(* PLC project extended wxHMI example, Unknown Beremiz 1 *)
(* stored: creationDateTime 2012-09-12T23:30:19, modificationDateTime 2018-09-26T14:07:02 *)

FUNCTION_BLOCK clock
  VAR
    TimerOn : TON;
  END_VAR
  VAR_OUTPUT
    Out : BOOL;
  END_VAR
  VAR_INPUT
    Period : TIME := T#3s;
  END_VAR
  VAR
    TimerOff : TON;
  END_VAR
  VAR  (* added by the conversion: wires and edge detectors of the diagram *)
    _DIV16_OUT : TIME;
  END_VAR

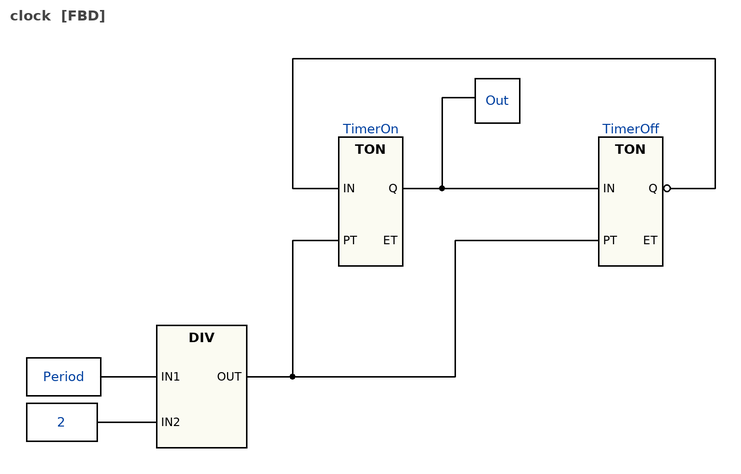
(* FBD diagram, written out as Structured Text *)
_DIV16_OUT := Period / 2;
TimerOff(IN := TimerOn.Q, PT := _DIV16_OUT);
TimerOn(IN := NOT TimerOff.Q, PT := _DIV16_OUT);
Out := TimerOn.Q;
END_FUNCTION_BLOCK

FUNCTION_BLOCK axis
  VAR_INPUT
    Power : BOOL;
    Up : BOOL;
    Down : BOOL;
  END_VAR
  VAR_OUTPUT
    Out : INT;
  END_VAR
  VAR
    axis_conuter : CTUD;
    clock0 : clock;
  END_VAR
  VAR  (* added by the conversion: wires and edge detectors of the diagram *)
    _AND4_OUT : BOOL;
    R_TRIG1 : R_TRIG;
    R_TRIG2 : R_TRIG;
  END_VAR

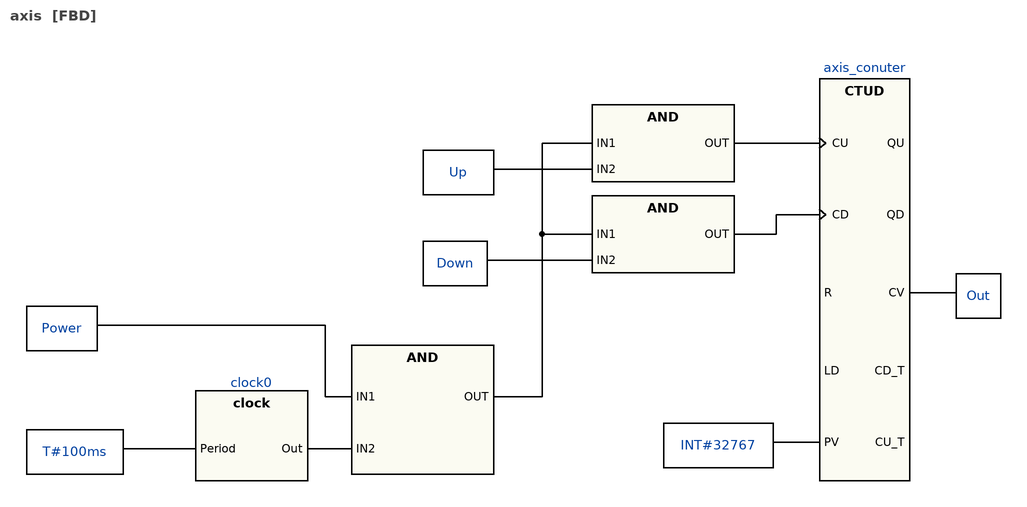
(* FBD diagram, written out as Structured Text *)
clock0(Period := T#100ms);
_AND4_OUT := Power AND clock0.Out;
R_TRIG1(CLK := _AND4_OUT AND Up);
R_TRIG2(CLK := _AND4_OUT AND Down);
axis_conuter(CU := R_TRIG1.Q, CD := R_TRIG2.Q, PV := INT#32767);
Out := axis_conuter.CV;
END_FUNCTION_BLOCK

PROGRAM main
  VAR_EXTERNAL
    Power_ON : BOOL;
    Power_OFF : BOOL;
  END_VAR
  VAR
    power : BOOL;
  END_VAR
  VAR_EXTERNAL
    DrawTest : BOOL;
    DrawTestBtn : BOOL;
    DrawLogo : BOOL;
    XaxisPos : INT;
    YaxisPos : INT;
    ZaxisPos : INT;
    TaxisPos : INT;
  END_VAR
  VAR
    PowerCtrl : RS;
    Xaxis : axis;
  END_VAR
  VAR_EXTERNAL
    XAxisMinus : BOOL;
    XAxisPlus : BOOL;
    YAxisPlus : BOOL;
    YAxisMinus : BOOL;
    ZAxisPlus : BOOL;
    ZAxisMinus : BOOL;
    TAxisPlus : BOOL;
    TAxisMinus : BOOL;
  END_VAR
  VAR
    Yaxis : axis;
    Taxis : axis;
    Zaxis : axis;
    DrawTestDo : RS;
    DrawLogoDo : RS;
  END_VAR

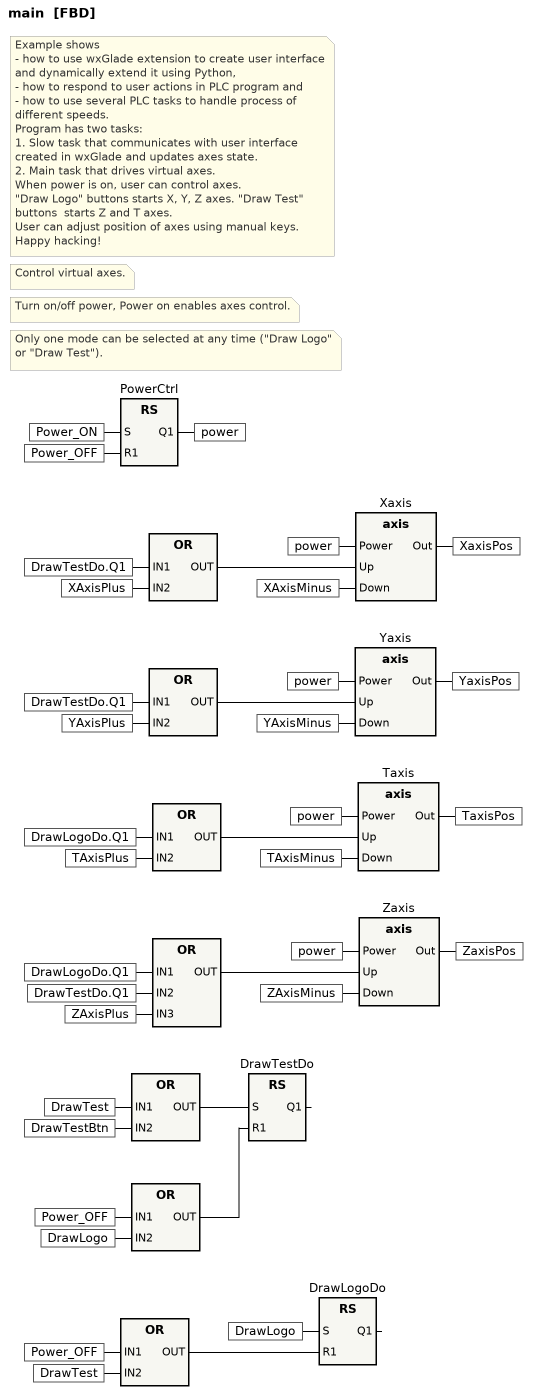
(* FBD diagram, written out as Structured Text *)
(* Example shows 
- how to use wxGlade extension to create user interface and dynamically extend it using Python, 
- how to respond to user actions in PLC program and 
- how to use several PLC tasks to handle process of different speeds.

Program has two tasks:
1. Slow task that communicates with user interface created in wxGlade and updates axes state.
2. Main task that drives virtual axes.

When power is on, user can control axes.
"Draw Logo" buttons starts X, Y, Z axes. "Draw Test" buttons  starts Z and T axes. 
User can adjust position of axes using manual keys.


Happy hacking! *)
(* Turn on/off power, Power on enables axes control. *)
PowerCtrl(S := Power_ON, R1 := Power_OFF);
power := PowerCtrl.Q1;
(* Only one mode can be selected at any time ("Draw Logo" or "Draw Test"). *)
(* Control virtual axes. *)
Xaxis(Power := power, Up := DrawTestDo.Q1 OR XAxisPlus, Down := XAxisMinus);
XaxisPos := Xaxis.Out;
Yaxis(Power := power, Up := DrawTestDo.Q1 OR YAxisPlus, Down := YAxisMinus);
YaxisPos := Yaxis.Out;
Zaxis(Power := power, Up := DrawLogoDo.Q1 OR DrawTestDo.Q1 OR ZAxisPlus, Down := ZAxisMinus);
ZaxisPos := Zaxis.Out;
Taxis(Power := power, Up := DrawLogoDo.Q1 OR TAxisPlus, Down := TAxisMinus);
TaxisPos := Taxis.Out;
DrawTestDo(S := DrawTest OR DrawTestBtn, R1 := Power_OFF OR DrawLogo);
DrawLogoDo(S := DrawLogo, R1 := Power_OFF OR DrawTest);
END_PROGRAM

PROGRAM ReadGUIdata
  VAR
    python_poll0 : python_poll;
  END_VAR

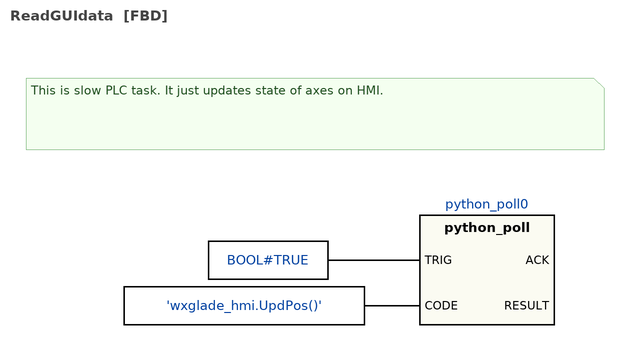
(* FBD diagram, written out as Structured Text *)
(* This is slow PLC task. It just updates state of axes on HMI. *)
python_poll0(TRIG := BOOL#TRUE, CODE := 'wxglade_hmi.UpdPos()');
END_PROGRAM

PROGRAM Declarations
  VAR
    InitValue : DINT := 17;
    NotInitializedVariable : DINT;
    counter : DINT;
  END_VAR

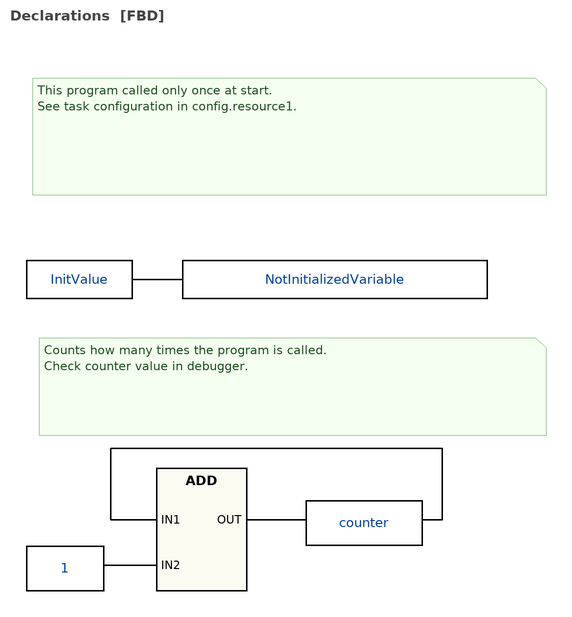
(* FBD diagram, written out as Structured Text *)
(* This program called only once at start.
See task configuration in config.resource1. *)
NotInitializedVariable := InitValue;
(* Counts how many times the program is called.
Check counter value in debugger. *)
counter := counter + 1;
END_PROGRAM

CONFIGURATION config
  RESOURCE resource1 ON PLC
    VAR_GLOBAL
      Initialize : BOOL := TRUE;
    END_VAR
    TASK InitOneShot(SINGLE := Initialize, PRIORITY := 0);
    TASK ControlTask(INTERVAL := T#2ms, PRIORITY := 1);
    TASK GUIupdate(INTERVAL := T#200ms, PRIORITY := 0);
    PROGRAM Initializer WITH InitOneShot : Declarations;
    PROGRAM MainInstance WITH ControlTask : main;
    PROGRAM PosReader WITH GUIupdate : ReadGUIdata;
  END_RESOURCE
END_CONFIGURATION
